{attribute 'qualified_only'}
VAR_GLOBAL
	axis1 : Tc2_MC2.AXIS_REF;
END_VAR

(* stored: Version 1.1.0.1, ProductVersion 3.1.4024.11
   GVL GVL: Id {5fc3267b-0f40-4fc4-b6cf-9bdcbc491d1a} *)
